Fanuc KAREL source: DELETE_NODE.kl

PROGRAM T
%NOLOCKGROUP
VAR
 v0 : PATH
 v1 : INTEGER
 v2 : INTEGER
BEGIN
 DELETE_NODE(v0, v1, v2)
END T
